Fanuc KAREL source: kb00096.KL

PROGRAM KB00096
%NOLOCKGROUP
VAR
P1:INTEGER;P2:INTEGER;P3:INTEGER;P4:REAL;P5 : STRING[80];P6:INTEGER
BEGIN
--
--
--
--
--
P1=1
P2=1
P3=1
P4=1.0
P5='A'
P6=1
GET_TPE_PRM(P1,P2,P3,P4,P5,P6)
END KB00096
